// TIA Portal V16 export
// export: Created 2023-07-30T20:35:42.4261995Z, ExportSetting WithDefaults, DisplayName Totally Integrated Automation Portal, DisplayVersion V16, DisplayName TIA Portal Version Control Interface, DisplayVersion V16, DisplayName TIA Portal Openness, DisplayVersion V16, DisplayName STEP 7 Professional, DisplayVersion V16, DisplayName STEP 7 Safety, DisplayVersion V16, DisplayName WinCC Professional, DisplayVersion V16
DATA_BLOCK "connect"   // DB4
{ S7_Optimized_Access := 'TRUE' }
VERSION : 0.1
// stored: AutoNumber true, DBAccessibleFromOPCUA true, IsOnlyStoredInLoadMemory false, IsRetainMemResEnabled false, IsWriteProtectedInAS false, MemoryReserve 100
   VAR
      req : Bool;
      disconnect : Bool;
      send { S7_SetPoint := 'True'} : TCON_IP_v4;
      recv : TCON_IP_v4;
   END_VAR
BEGIN
   send.InterfaceId := 64;
   send.ID := 1;
   send.ConnectionType := 11;
   send.ActiveEstablished := true;
   send.RemoteAddress.ADDR[1] := 192;
   send.RemoteAddress.ADDR[2] := 168;
   send.RemoteAddress.ADDR[3] := 1;
   send.RemoteAddress.ADDR[4] := 11;
   send.RemotePort := 502;
   send.LocalPort := 502;
   recv.InterfaceId := 64;
   recv.ID := 2;
   recv.ConnectionType := 11;
   recv.ActiveEstablished := true;
   recv.RemoteAddress.ADDR[1] := 192;
   recv.RemoteAddress.ADDR[2] := 168;
   recv.RemoteAddress.ADDR[3] := 1;
   recv.RemoteAddress.ADDR[4] := 11;
   recv.RemotePort := 502;
   recv.LocalPort := 502;
END_DATA_BLOCK
